FUNCTION F_Concat7_Large : STRING(StringsParams.MAX_STRING_LENGTH)
VAR_IN_OUT CONSTANT
	sOne : STRING(StringsParams.MAX_STRING_LENGTH);
	sTwo : STRING(StringsParams.MAX_STRING_LENGTH);
	sThree : STRING(StringsParams.MAX_STRING_LENGTH);
	sFour : STRING(StringsParams.MAX_STRING_LENGTH);
	sFive : STRING(StringsParams.MAX_STRING_LENGTH);
	sSix : STRING(StringsParams.MAX_STRING_LENGTH);
	sSeven : STRING(StringsParams.MAX_STRING_LENGTH);
END_VAR
VAR
	str : STRING(StringsParams.MAX_STRING_LENGTH);
END_VAR

str := F_Concat6_Large( sTwo, sThree, sFour, sFive, sSix, sSeven);
F_Concat7_Large := 
	F_ConcatLarge(
		sOne,
		str
	);

END_FUNCTION

(* stored: Version 1.1.0.1, ProductVersion 3.1.4022.6
   POU F_Concat7_Large: Id {55de9d64-fb93-4bfb-95dd-a0921848ec99}, SpecialFunc None *)
